TYPE InputBase_8311D824 :
STRUCT
END_STRUCT
END_TYPE

(* stored: Version 1.2.0.0, ProductVersion 3.1.4024.11
   DUT InputBase_8311D824: Id {589ab15b-8552-41da-b6d2-26d183a03d89} *)
